PROGRAM MAIN
VAR
	i : INT;
	bTestMqtt : BOOL;
	fbMqtt : FB_TestMqtt;
	bTestHttp : BOOL := TRUE;
	fbHttp : FB_TestHTTP;
	
END_VAR

i := i + 1;

IF bTestMqtt THEN
	fbMqtt();	
END_IF
IF bTestHttp THEN
	fbHttp();	
END_IF

END_PROGRAM

(* stored: Version 1.1.0.1, ProductVersion 3.1.4024.0
   POU MAIN: Id {cded3529-4d1e-4b4f-a3db-0d3c1cd5c7c2}, SpecialFunc None *)
